TYPE ST_P_RELEASE_MRT :
STRUCT
END_STRUCT
END_TYPE

(* stored: Version 1.1.0.1, ProductVersion 3.1.4024.10
   DUT ST_P_RELEASE_MRT: Id {ee5a98ef-6852-4225-87fa-f5038b331c3d} *)
